PROGRAM MAIN
VAR
	//alias
	_HRESULT_TestSuite : _HRESULT_TestSuite;
    _FLOAT_TestSuite : _FLOAT_TestSuite;
	
	// primitive
	_BOOL_TestSuite : _BOOL_TestSuite;
    _BYTE_TestSuite : _BYTE_TestSuite;
    _WORD_TestSuite : _WORD_TestSuite;
    _DWORD_TestSuite : _DWORD_TestSuite;
    _LWORD_TestSuite : _LWORD_TestSuite;
    
    _SINT_TestSuite : _SINT_TestSuite;
    _INT_TestSuite : _INT_TestSuite;
    _DINT_TestSuite : _DINT_TestSuite;
    _LINT_TestSuite : _LINT_TestSuite;
    
    _USINT_TestSuite : _USINT_TestSuite;
    _UINT_TestSuite : _UINT_TestSuite;
    _UDINT_TestSuite : _UDINT_TestSuite;
    _ULINT_TestSuite : _ULINT_TestSuite;
    
    _REAL_TestSuite : _REAL_TestSuite;
    _LREAL_TestSuite : _LREAL_TestSuite;
    
    //_TIME_TestSuite : _TIME_TestSuite;
    //_LTIME_TestSuite : _LTIME_TestSuite;
    _TOD_TestSuite : _TOD_TestSuite;
    _TIME_OF_DAY_TestSuite : _TIME_OF_DAY_TestSuite;
    
    //_DATE_TestSuite : _TIME_TestSuite;
    //_DATE_AND_TIME_TestSuite : _DATE_AND_TIME_TestSuite;
    _DT_TestSuite : _DT_TestSuite;
    
    //_LDATE, LDATE_AND_TIME, _LDT, LTIME_OF_DAY & _LTOD require TC build >=4026.0
	
	// struct
	_TIMESTRUCT_TestSuite : _TIMESTRUCT_TestSuite;
END_VAR

TcUnit.RUN();

END_PROGRAM

(* stored: Version 1.1.0.1, ProductVersion 3.1.4024.12
   POU MAIN: Id {7bf63626-4b20-4fda-b93b-546e8359a2c5}, SpecialFunc None *)
